FUNCTION_BLOCK Motor_Notimplemented
VAR_INPUT
END_VAR
VAR_OUTPUT
END_VAR
VAR
END_VAR

END_FUNCTION_BLOCK

(* stored: Version 1.1.0.1, ProductVersion 3.1.4024.6
   POU Motor_Notimplemented: Id {7d4abe09-fc4f-42ac-9265-2a154e6bbf0e}, SpecialFunc None *)
